	//Alarm Priority setpoint
	{attribute 'OPC.UA.DA' :='1'}
	popa_0082_pt_3119_b_low_priority : INT;
	//Alarm delay setpoint(seconds)
	{attribute 'OPC.UA.DA' :='1'}
	popa_0082_pt_3119_b_low_delay_setpoint : INT;
	//Alarm active for HMI
	{attribute 'OPC.UA.DA' :='1'}
	popa_0082_pt_3119_b_low_active : BOOL;
	//Analog Alarm Setpoint
	{attribute 'OPC.UA.DA' :='1'}
	popa_0082_pt_3119_b_low_setpoint : REAL;
	//Alarm enable
	{attribute 'OPC.UA.DA' :='1'}
	popa_0082_pt_3119_b_low_enable: BOOL;
	
	//Alarm Priority setpoint
	{attribute 'OPC.UA.DA' :='1'}
	popa_0082_pt_3119_b_high_priority : INT;
	//Alarm delay setpoint(seconds)
	{attribute 'OPC.UA.DA' :='1'}
	popa_0082_pt_3119_b_high_delay_setpoint : INT;
	//Alarm active for HMI
	{attribute 'OPC.UA.DA' :='1'}
	popa_0082_pt_3119_b_high_active : BOOL;
	//Analog Alarm Setpoint
	{attribute 'OPC.UA.DA' :='1'}
	popa_0082_pt_3119_b_high_setpoint : REAL;
	//Alarm enable
	{attribute 'OPC.UA.DA' :='1'}
	popa_0082_pt_3119_b_high_enable: BOOL;
	
	//Alarm Priority setpoint
	{attribute 'OPC.UA.DA' :='1'}
	popa_0082_pt_3119_b_high_high_priority : INT;
	//Alarm delay setpoint(seconds)
	{attribute 'OPC.UA.DA' :='1'}
	popa_0082_pt_3119_b_high_high_delay_setpoint : INT;
	//Alarm active for HMI
	{attribute 'OPC.UA.DA' :='1'}
	popa_0082_pt_3119_b_high_high_active : BOOL;
	//Analog Alarm Setpoint
	{attribute 'OPC.UA.DA' :='1'}
	popa_0082_pt_3119_b_high_high_setpoint : REAL;
	//Alarm enable
	{attribute 'OPC.UA.DA' :='1'}
	popa_0082_pt_3119_b_high_high_enable: BOOL;
	
	
	//Raw Min value for analog input
	{attribute 'OPC.UA.DA' :='1'}
	popa_0082_pt_3119_b_raw_min : REAL :=0;
	//Raw max value for analog input
	{attribute 'OPC.UA.DA' :='1'}
	popa_0082_pt_3119_b_raw_max : REAL :=32767;
	//EU Min value for analog input
	{attribute 'OPC.UA.DA' :='1'}
	popa_0082_pt_3119_b_eu_min : REAL;
	//EU Max value for analog input
	{attribute 'OPC.UA.DA' :='1'}
	popa_0082_pt_3119_b_eu_max : REAL;
	//Filter factor value for analog input
	{attribute 'OPC.UA.DA' :='1'}
	popa_0082_pt_3119_b_filter_factor : REAL;
	//Scaled value for analog input
	{attribute 'OPC.UA.DA' :='1'}
	popa_0082_pt_3119_b_scaled_value : REAL;
	
	//---pt_3219-----------------------------------------------------------------------------------------------------------------------
	//Alarm Priority setpoint
	{attribute 'OPC.UA.DA' :='1'}
	popa_0082_pt_3219_b_low_low_priority : INT;
	//Alarm delay setpoint(seconds)
	{attribute 'OPC.UA.DA' :='1'}
	popa_0082_pt_3219_b_low_low_delay_setpoint : INT;
	//Alarm active for HMI
	{attribute 'OPC.UA.DA' :='1'}
	popa_0082_pt_3219_b_low_low_active : BOOL;
	//Analog Alarm Setpoint
	{attribute 'OPC.UA.DA' :='1'}
	popa_0082_pt_3219_b_low_low_setpoint : REAL;
	//Alarm enable
	{attribute 'OPC.UA.DA' :='1'}
	popa_0082_pt_3219_b_low_low_enable: BOOL;
	
	//Alarm Priority setpoint
	{attribute 'OPC.UA.DA' :='1'}
	popa_0082_pt_3219_b_low_priority : INT;
	//Alarm delay setpoint(seconds)
	{attribute 'OPC.UA.DA' :='1'}
	popa_0082_pt_3219_b_low_delay_setpoint : INT;
	//Alarm active for HMI
	{attribute 'OPC.UA.DA' :='1'}
	popa_0082_pt_3219_b_low_active : BOOL;
	//Analog Alarm Setpoint
	{attribute 'OPC.UA.DA' :='1'}
	popa_0082_pt_3219_b_low_setpoint : REAL;
	//Alarm enable
	{attribute 'OPC.UA.DA' :='1'}
	popa_0082_pt_3219_b_low_enable: BOOL;
	
	//Alarm Priority setpoint
	{attribute 'OPC.UA.DA' :='1'}
	popa_0082_pt_3219_b_high_priority : INT;
	//Alarm delay setpoint(seconds)
	{attribute 'OPC.UA.DA' :='1'}
	popa_0082_pt_3219_b_high_delay_setpoint : INT;
	//Alarm active for HMI
	{attribute 'OPC.UA.DA' :='1'}
	popa_0082_pt_3219_b_high_active : BOOL;
	//Analog Alarm Setpoint
	{attribute 'OPC.UA.DA' :='1'}
	popa_0082_pt_3219_b_high_setpoint : REAL;
	//Alarm enable
	{attribute 'OPC.UA.DA' :='1'}
	popa_0082_pt_3219_b_high_enable: BOOL;
	
	//Alarm Priority setpoint
	{attribute 'OPC.UA.DA' :='1'}
	popa_0082_pt_3219_b_high_high_priority : INT;
	//Alarm delay setpoint(seconds)
	{attribute 'OPC.UA.DA' :='1'}
	popa_0082_pt_3219_b_high_high_delay_setpoint : INT;
	//Alarm active for HMI
	{attribute 'OPC.UA.DA' :='1'}
	popa_0082_pt_3219_b_high_high_active : BOOL;
	//Analog Alarm Setpoint
	{attribute 'OPC.UA.DA' :='1'}
	popa_0082_pt_3219_b_high_high_setpoint : REAL;
	//Alarm enable
	{attribute 'OPC.UA.DA' :='1'}
	popa_0082_pt_3219_b_high_high_enable: BOOL;
	
	
	//Raw Min value for analog input
	{attribute 'OPC.UA.DA' :='1'}
	popa_0082_pt_3219_b_raw_min : REAL :=0;
	//Raw max value for analog input
	{attribute 'OPC.UA.DA' :='1'}
	popa_0082_pt_3219_b_raw_max : REAL :=32767;
	//EU Min value for analog input
	{attribute 'OPC.UA.DA' :='1'}
	popa_0082_pt_3219_b_eu_min : REAL;
	//EU Max value for analog input
	{attribute 'OPC.UA.DA' :='1'}
	popa_0082_pt_3219_b_eu_max : REAL;
	//Filter factor value for analog input
	{attribute 'OPC.UA.DA' :='1'}
	popa_0082_pt_3219_b_filter_factor : REAL;
	//Scaled value for analog input
	{attribute 'OPC.UA.DA' :='1'}
	popa_0082_pt_3219_b_scaled_value : REAL;
	
	//---pt_3319-----------------------------------------------------------------------------------------------------------------------
	//Alarm Priority setpoint
	{attribute 'OPC.UA.DA' :='1'}
	popa_0082_pt_3319_b_low_low_priority : INT;
	//Alarm delay setpoint(seconds)
	{attribute 'OPC.UA.DA' :='1'}
	popa_0082_pt_3319_b_low_low_delay_setpoint : INT;
	//Alarm active for HMI
	{attribute 'OPC.UA.DA' :='1'}
	popa_0082_pt_3319_b_low_low_active : BOOL;
	//Analog Alarm Setpoint
	{attribute 'OPC.UA.DA' :='1'}
	popa_0082_pt_3319_b_low_low_setpoint : REAL;
	//Alarm enable
	{attribute 'OPC.UA.DA' :='1'}
	popa_0082_pt_3319_b_low_low_enable: BOOL;
	
	//Alarm Priority setpoint
	{attribute 'OPC.UA.DA' :='1'}
	popa_0082_pt_3319_b_low_priority : INT;
	//Alarm delay setpoint(seconds)
	{attribute 'OPC.UA.DA' :='1'}
	popa_0082_pt_3319_b_low_delay_setpoint : INT;
	//Alarm active for HMI
	{attribute 'OPC.UA.DA' :='1'}
	popa_0082_pt_3319_b_low_active : BOOL;
	//Analog Alarm Setpoint
	{attribute 'OPC.UA.DA' :='1'}
	popa_0082_pt_3319_b_low_setpoint : REAL;
	//Alarm enable
	{attribute 'OPC.UA.DA' :='1'}
	popa_0082_pt_3319_b_low_enable: BOOL;
	
	//Alarm Priority setpoint
	{attribute 'OPC.UA.DA' :='1'}
	popa_0082_pt_3319_b_high_priority : INT;
	//Alarm delay setpoint(seconds)
	{attribute 'OPC.UA.DA' :='1'}
	popa_0082_pt_3319_b_high_delay_setpoint : INT;
	//Alarm active for HMI
	{attribute 'OPC.UA.DA' :='1'}
	popa_0082_pt_3319_b_high_active : BOOL;
	//Analog Alarm Setpoint
	{attribute 'OPC.UA.DA' :='1'}
	popa_0082_pt_3319_b_high_setpoint : REAL;
	//Alarm enable
	{attribute 'OPC.UA.DA' :='1'}
	popa_0082_pt_3319_b_high_enable: BOOL;
	
	//Alarm Priority setpoint
	{attribute 'OPC.UA.DA' :='1'}
	popa_0082_pt_3319_b_high_high_priority : INT;
	//Alarm delay setpoint(seconds)
	{attribute 'OPC.UA.DA' :='1'}
	popa_0082_pt_3319_b_high_high_delay_setpoint : INT;
	//Alarm active for HMI
	{attribute 'OPC.UA.DA' :='1'}
	popa_0082_pt_3319_b_high_high_active : BOOL;
	//Analog Alarm Setpoint
	{attribute 'OPC.UA.DA' :='1'}
	popa_0082_pt_3319_b_high_high_setpoint : REAL;
	//Alarm enable
	{attribute 'OPC.UA.DA' :='1'}
	popa_0082_pt_3319_b_high_high_enable: BOOL;
	
	
	//Raw Min value for analog input
	{attribute 'OPC.UA.DA' :='1'}
	popa_0082_pt_3319_b_raw_min : REAL :=0;
	//Raw max value for analog input
	{attribute 'OPC.UA.DA' :='1'}
	popa_0082_pt_3319_b_raw_max : REAL :=32767;
	//EU Min value for analog input
	{attribute 'OPC.UA.DA' :='1'}
	popa_0082_pt_3319_b_eu_min : REAL;
	//EU Max value for analog input
	{attribute 'OPC.UA.DA' :='1'}
	popa_0082_pt_3319_b_eu_max : REAL;
	//Filter factor value for analog input
	{attribute 'OPC.UA.DA' :='1'}
	popa_0082_pt_3319_b_filter_factor : REAL;
	//Scaled value for analog input
	{attribute 'OPC.UA.DA' :='1'}
	popa_0082_pt_3319_b_scaled_value : REAL;
	
	//---pt_3141-----------------------------------------------------------------------------------------------------------------------
	//Alarm Priority setpoint
	{attribute 'OPC.UA.DA' :='1'}
	popa_0082_pt_3141_b_low_low_priority : INT;
	//Alarm delay setpoint(seconds)
	{attribute 'OPC.UA.DA' :='1'}
	popa_0082_pt_3141_b_low_low_delay_setpoint : INT;
	//Alarm active for HMI
	{attribute 'OPC.UA.DA' :='1'}
	popa_0082_pt_3141_b_low_low_active : BOOL;
	//Analog Alarm Setpoint
	{attribute 'OPC.UA.DA' :='1'}
	popa_0082_pt_3141_b_low_low_setpoint : REAL;
	//Alarm enable
	{attribute 'OPC.UA.DA' :='1'}
	popa_0082_pt_3141_b_low_low_enable: BOOL;
	
	//Alarm Priority setpoint
	{attribute 'OPC.UA.DA' :='1'}
	popa_0082_pt_3141_b_low_priority : INT;
	//Alarm delay setpoint(seconds)
	{attribute 'OPC.UA.DA' :='1'}
	popa_0082_pt_3141_b_low_delay_setpoint : INT;
	//Alarm active for HMI
	{attribute 'OPC.UA.DA' :='1'}
	popa_0082_pt_3141_b_low_active : BOOL;
	//Analog Alarm Setpoint
	{attribute 'OPC.UA.DA' :='1'}
	popa_0082_pt_3141_b_low_setpoint : REAL;
	//Alarm enable
	{attribute 'OPC.UA.DA' :='1'}
	popa_0082_pt_3141_b_low_enable: BOOL;
	
	//Alarm Priority setpoint
	{attribute 'OPC.UA.DA' :='1'}
	popa_0082_pt_3141_b_high_priority : INT;
	//Alarm delay setpoint(seconds)
	{attribute 'OPC.UA.DA' :='1'}
	popa_0082_pt_3141_b_high_delay_setpoint : INT;
	//Alarm active for HMI
	{attribute 'OPC.UA.DA' :='1'}
	popa_0082_pt_3141_b_high_active : BOOL;
	//Analog Alarm Setpoint
	{attribute 'OPC.UA.DA' :='1'}
	popa_0082_pt_3141_b_high_setpoint : REAL;
	//Alarm enable
	{attribute 'OPC.UA.DA' :='1'}
	popa_0082_pt_3141_b_high_enable: BOOL;
	
	//Alarm Priority setpoint
	{attribute 'OPC.UA.DA' :='1'}
	popa_0082_pt_3141_b_high_high_priority : INT;
	//Alarm delay setpoint(seconds)
	{attribute 'OPC.UA.DA' :='1'}
	popa_0082_pt_3141_b_high_high_delay_setpoint : INT;
	//Alarm active for HMI
	{attribute 'OPC.UA.DA' :='1'}
	popa_0082_pt_3141_b_high_high_active : BOOL;
	//Analog Alarm Setpoint
	{attribute 'OPC.UA.DA' :='1'}
	popa_0082_pt_3141_b_high_high_setpoint : REAL;
	//Alarm enable
	{attribute 'OPC.UA.DA' :='1'}
	popa_0082_pt_3141_b_high_high_enable: BOOL;
	
	
	//Raw Min value for analog input
	{attribute 'OPC.UA.DA' :='1'}
	popa_0082_pt_3141_b_raw_min : REAL :=0;
	//Raw max value for analog input
	{attribute 'OPC.UA.DA' :='1'}
	popa_0082_pt_3141_b_raw_max : REAL :=32767;
	//EU Min value for analog input
	{attribute 'OPC.UA.DA' :='1'}
	popa_0082_pt_3141_b_eu_min : REAL;
	//EU Max value for analog input
	{attribute 'OPC.UA.DA' :='1'}
	popa_0082_pt_3141_b_eu_max : REAL;
	//Filter factor value for analog input
	{attribute 'OPC.UA.DA' :='1'}
	popa_0082_pt_3141_b_filter_factor : REAL;
	//Scaled value for analog input
	{attribute 'OPC.UA.DA' :='1'}
	popa_0082_pt_3141_b_scaled_value : REAL;
	
	//---pt_3241-----------------------------------------------------------------------------------------------------------------------
	//Alarm Priority setpoint
	{attribute 'OPC.UA.DA' :='1'}
	popa_0082_pt_3241_b_low_low_priority : INT;
	//Alarm delay setpoint(seconds)
	{attribute 'OPC.UA.DA' :='1'}
	popa_0082_pt_3241_b_low_low_delay_setpoint : INT;
	//Alarm active for HMI
	{attribute 'OPC.UA.DA' :='1'}
	popa_0082_pt_3241_b_low_low_active : BOOL;
	//Analog Alarm Setpoint
	{attribute 'OPC.UA.DA' :='1'}
	popa_0082_pt_3241_b_low_low_setpoint : REAL;
	//Alarm enable
	{attribute 'OPC.UA.DA' :='1'}
	popa_0082_pt_3241_b_low_low_enable: BOOL;
	
	//Alarm Priority setpoint
	{attribute 'OPC.UA.DA' :='1'}
	popa_0082_pt_3241_b_low_priority : INT;
	//Alarm delay setpoint(seconds)
	{attribute 'OPC.UA.DA' :='1'}
	popa_0082_pt_3241_b_low_delay_setpoint : INT;
	//Alarm active for HMI
	{attribute 'OPC.UA.DA' :='1'}
	popa_0082_pt_3241_b_low_active : BOOL;
	//Analog Alarm Setpoint
	{attribute 'OPC.UA.DA' :='1'}
	popa_0082_pt_3241_b_low_setpoint : REAL;
	//Alarm enable
	{attribute 'OPC.UA.DA' :='1'}
	popa_0082_pt_3241_b_low_enable: BOOL;
	
	//Alarm Priority setpoint
	{attribute 'OPC.UA.DA' :='1'}
	popa_0082_pt_3241_b_high_priority : INT;
	//Alarm delay setpoint(seconds)
	{attribute 'OPC.UA.DA' :='1'}
	popa_0082_pt_3241_b_high_delay_setpoint : INT;
	//Alarm active for HMI
	{attribute 'OPC.UA.DA' :='1'}
	popa_0082_pt_3241_b_high_active : BOOL;
	//Analog Alarm Setpoint
	{attribute 'OPC.UA.DA' :='1'}
	popa_0082_pt_3241_b_high_setpoint : REAL;
	//Alarm enable
	{attribute 'OPC.UA.DA' :='1'}
	popa_0082_pt_3241_b_high_enable: BOOL;
	
	//Alarm Priority setpoint
	{attribute 'OPC.UA.DA' :='1'}
	popa_0082_pt_3241_b_high_high_priority : INT;
	//Alarm delay setpoint(seconds)
	{attribute 'OPC.UA.DA' :='1'}
	popa_0082_pt_3241_b_high_high_delay_setpoint : INT;
	//Alarm active for HMI
	{attribute 'OPC.UA.DA' :='1'}
	popa_0082_pt_3241_b_high_high_active : BOOL;
	//Analog Alarm Setpoint
	{attribute 'OPC.UA.DA' :='1'}
	popa_0082_pt_3241_b_high_high_setpoint : REAL;
	//Alarm enable
	{attribute 'OPC.UA.DA' :='1'}
	popa_0082_pt_3241_b_high_high_enable: BOOL;
	
	
	//Raw Min value for analog input
	{attribute 'OPC.UA.DA' :='1'}
	popa_0082_pt_3241_b_raw_min : REAL :=0;
	//Raw max value for analog input
	{attribute 'OPC.UA.DA' :='1'}
	popa_0082_pt_3241_b_raw_max : REAL :=32767;
	//EU Min value for analog input
	{attribute 'OPC.UA.DA' :='1'}
	popa_0082_pt_3241_b_eu_min : REAL;
	//EU Max value for analog input
	{attribute 'OPC.UA.DA' :='1'}
	popa_0082_pt_3241_b_eu_max : REAL;
	//Filter factor value for analog input
	{attribute 'OPC.UA.DA' :='1'}
	popa_0082_pt_3241_b_filter_factor : REAL;
	//Scaled value for analog input
	{attribute 'OPC.UA.DA' :='1'}
	popa_0082_pt_3241_b_scaled_value : REAL;
	
	//---pt_3341-----------------------------------------------------------------------------------------------------------------------
	//Alarm Priority setpoint
	{attribute 'OPC.UA.DA' :='1'}
	popa_0082_pt_3341_b_low_low_priority : INT;
	//Alarm delay setpoint(seconds)
	{attribute 'OPC.UA.DA' :='1'}
	popa_0082_pt_3341_b_low_low_delay_setpoint : INT;
	//Alarm active for HMI
	{attribute 'OPC.UA.DA' :='1'}
	popa_0082_pt_3341_b_low_low_active : BOOL;
	//Analog Alarm Setpoint
	{attribute 'OPC.UA.DA' :='1'}
	popa_0082_pt_3341_b_low_low_setpoint : REAL;
	//Alarm enable
	{attribute 'OPC.UA.DA' :='1'}
	popa_0082_pt_3341_b_low_low_enable: BOOL;
	
	//Alarm Priority setpoint
	{attribute 'OPC.UA.DA' :='1'}
	popa_0082_pt_3341_b_low_priority : INT;
	//Alarm delay setpoint(seconds)
	{attribute 'OPC.UA.DA' :='1'}
	popa_0082_pt_3341_b_low_delay_setpoint : INT;
	//Alarm active for HMI
	{attribute 'OPC.UA.DA' :='1'}
	popa_0082_pt_3341_b_low_active : BOOL;
	//Analog Alarm Setpoint
	{attribute 'OPC.UA.DA' :='1'}
	popa_0082_pt_3341_b_low_setpoint : REAL;
	//Alarm enable
	{attribute 'OPC.UA.DA' :='1'}
	popa_0082_pt_3341_b_low_enable: BOOL;
	
	//Alarm Priority setpoint
	{attribute 'OPC.UA.DA' :='1'}
	popa_0082_pt_3341_b_high_priority : INT;
	//Alarm delay setpoint(seconds)
	{attribute 'OPC.UA.DA' :='1'}
	popa_0082_pt_3341_b_high_delay_setpoint : INT;
	//Alarm active for HMI
	{attribute 'OPC.UA.DA' :='1'}
	popa_0082_pt_3341_b_high_active : BOOL;
	//Analog Alarm Setpoint
	{attribute 'OPC.UA.DA' :='1'}
	popa_0082_pt_3341_b_high_setpoint : REAL;
	//Alarm enable
	{attribute 'OPC.UA.DA' :='1'}
	popa_0082_pt_3341_b_high_enable: BOOL;
	
	//Alarm Priority setpoint
	{attribute 'OPC.UA.DA' :='1'}
	popa_0082_pt_3341_b_high_high_priority : INT;
	//Alarm delay setpoint(seconds)
	{attribute 'OPC.UA.DA' :='1'}
	popa_0082_pt_3341_b_high_high_delay_setpoint : INT;
	//Alarm active for HMI
	{attribute 'OPC.UA.DA' :='1'}
	popa_0082_pt_3341_b_high_high_active : BOOL;
	//Analog Alarm Setpoint
	{attribute 'OPC.UA.DA' :='1'}
	popa_0082_pt_3341_b_high_high_setpoint : REAL;
	//Alarm enable
	{attribute 'OPC.UA.DA' :='1'}
	popa_0082_pt_3341_b_high_high_enable: BOOL;
	
	
	//Raw Min value for analog input
	{attribute 'OPC.UA.DA' :='1'}
	popa_0082_pt_3341_b_raw_min : REAL :=0;
	//Raw max value for analog input
	{attribute 'OPC.UA.DA' :='1'}
	popa_0082_pt_3341_b_raw_max : REAL :=32767;
	//EU Min value for analog input
	{attribute 'OPC.UA.DA' :='1'}
	popa_0082_pt_3341_b_eu_min : REAL;
	//EU Max value for analog input
	{attribute 'OPC.UA.DA' :='1'}
	popa_0082_pt_3341_b_eu_max : REAL;
	//Filter factor value for analog input
	{attribute 'OPC.UA.DA' :='1'}
	popa_0082_pt_3341_b_filter_factor : REAL;
	//Scaled value for analog input
	{attribute 'OPC.UA.DA' :='1'}
	popa_0082_pt_3341_b_scaled_value : REAL;
	
//---pt_3428-----------------------------------------------------------------------------------------------------------------------
	//Alarm Priority setpoint
	{attribute 'OPC.UA.DA' :='1'}
	popa_0092_pt_3428_b_low_low_priority : INT;
	//Alarm delay setpoint(seconds)
	{attribute 'OPC.UA.DA' :='1'}
	popa_0092_pt_3428_b_low_low_delay_setpoint : INT;
	//Alarm active for HMI
	{attribute 'OPC.UA.DA' :='1'}
	popa_0092_pt_3428_b_low_low_active : BOOL;
	//Analog Alarm Setpoint
	{attribute 'OPC.UA.DA' :='1'}
	popa_0092_pt_3428_b_low_low_setpoint : REAL;
	//Alarm enable
	{attribute 'OPC.UA.DA' :='1'}
	popa_0092_pt_3428_b_low_low_enable: BOOL;
	
	//Alarm Priority setpoint
	{attribute 'OPC.UA.DA' :='1'}
	popa_0092_pt_3428_b_low_priority : INT;
	//Alarm delay setpoint(seconds)
	{attribute 'OPC.UA.DA' :='1'}
	popa_0092_pt_3428_b_low_delay_setpoint : INT;
	//Alarm active for HMI
	{attribute 'OPC.UA.DA' :='1'}
	popa_0092_pt_3428_b_low_active : BOOL;
	//Analog Alarm Setpoint
	{attribute 'OPC.UA.DA' :='1'}
	popa_0092_pt_3428_b_low_setpoint : REAL;
	//Alarm enable
	{attribute 'OPC.UA.DA' :='1'}
	popa_0092_pt_3428_b_low_enable: BOOL;
	
	//Alarm Priority setpoint
	{attribute 'OPC.UA.DA' :='1'}
	popa_0092_pt_3428_b_high_priority : INT;
	//Alarm delay setpoint(seconds)
	{attribute 'OPC.UA.DA' :='1'}
	popa_0092_pt_3428_b_high_delay_setpoint : INT;
	//Alarm active for HMI
	{attribute 'OPC.UA.DA' :='1'}
	popa_0092_pt_3428_b_high_active : BOOL;
	//Analog Alarm Setpoint
	{attribute 'OPC.UA.DA' :='1'}
	popa_0092_pt_3428_b_high_setpoint : REAL;
	//Alarm enable
	{attribute 'OPC.UA.DA' :='1'}
	popa_0092_pt_3428_b_high_enable: BOOL;
	
	//Alarm Priority setpoint
	{attribute 'OPC.UA.DA' :='1'}
	popa_0092_pt_3428_b_high_high_priority : INT;
	//Alarm delay setpoint(seconds)
	{attribute 'OPC.UA.DA' :='1'}
	popa_0092_pt_3428_b_high_high_delay_setpoint : INT;
	//Alarm active for HMI
	{attribute 'OPC.UA.DA' :='1'}
	popa_0092_pt_3428_b_high_high_active : BOOL;
	//Analog Alarm Setpoint
	{attribute 'OPC.UA.DA' :='1'}
	popa_0092_pt_3428_b_high_high_setpoint : REAL;
	//Alarm enable
	{attribute 'OPC.UA.DA' :='1'}
	popa_0092_pt_3428_b_high_high_enable: BOOL;
	
	
	//Raw Min value for analog input
	{attribute 'OPC.UA.DA' :='1'}
	popa_0092_pt_3428_b_raw_min : REAL :=0;
	//Raw max value for analog input
	{attribute 'OPC.UA.DA' :='1'}
	popa_0092_pt_3428_b_raw_max : REAL :=32767;
	//EU Min value for analog input
	{attribute 'OPC.UA.DA' :='1'}
	popa_0092_pt_3428_b_eu_min : REAL;
	//EU Max value for analog input
	{attribute 'OPC.UA.DA' :='1'}
	popa_0092_pt_3428_b_eu_max : REAL;
	//Filter factor value for analog input
	{attribute 'OPC.UA.DA' :='1'}
	popa_0092_pt_3428_b_filter_factor : REAL;
	//Scaled value for analog input
	{attribute 'OPC.UA.DA' :='1'}
	popa_0092_pt_3428_b_scaled_value : REAL;
	
	//---pt_3414-----------------------------------------------------------------------------------------------------------------------
	//Alarm Priority setpoint
	{attribute 'OPC.UA.DA' :='1'}
	popa_0092_pt_3414_b_low_low_priority : INT;
	//Alarm delay setpoint(seconds)
	{attribute 'OPC.UA.DA' :='1'}
	popa_0092_pt_3414_b_low_low_delay_setpoint : INT;
	//Alarm active for HMI
	{attribute 'OPC.UA.DA' :='1'}
	popa_0092_pt_3414_b_low_low_active : BOOL;
	//Analog Alarm Setpoint
	{attribute 'OPC.UA.DA' :='1'}
	popa_0092_pt_3414_b_low_low_setpoint : REAL;
	//Alarm enable
	{attribute 'OPC.UA.DA' :='1'}
	popa_0092_pt_3414_b_low_low_enable: BOOL;
	
	//Alarm Priority setpoint
	{attribute 'OPC.UA.DA' :='1'}
	popa_0092_pt_3414_b_low_priority : INT;
	//Alarm delay setpoint(seconds)
	{attribute 'OPC.UA.DA' :='1'}
	popa_0092_pt_3414_b_low_delay_setpoint : INT;
	//Alarm active for HMI
	{attribute 'OPC.UA.DA' :='1'}
	popa_0092_pt_3414_b_low_active : BOOL;
	//Analog Alarm Setpoint
	{attribute 'OPC.UA.DA' :='1'}
	popa_0092_pt_3414_b_low_setpoint : REAL;
	//Alarm enable
	{attribute 'OPC.UA.DA' :='1'}
	popa_0092_pt_3414_b_low_enable: BOOL;
	
	//Alarm Priority setpoint
	{attribute 'OPC.UA.DA' :='1'}
	popa_0092_pt_3414_b_high_priority : INT;
	//Alarm delay setpoint(seconds)
	{attribute 'OPC.UA.DA' :='1'}
	popa_0092_pt_3414_b_high_delay_setpoint : INT;
	//Alarm active for HMI
	{attribute 'OPC.UA.DA' :='1'}
	popa_0092_pt_3414_b_high_active : BOOL;
	//Analog Alarm Setpoint
	{attribute 'OPC.UA.DA' :='1'}
	popa_0092_pt_3414_b_high_setpoint : REAL;
	//Alarm enable
	{attribute 'OPC.UA.DA' :='1'}
	popa_0092_pt_3414_b_high_enable: BOOL;
	
	//Alarm Priority setpoint
	{attribute 'OPC.UA.DA' :='1'}
	popa_0092_pt_3414_b_high_high_priority : INT;
	//Alarm delay setpoint(seconds)
	{attribute 'OPC.UA.DA' :='1'}
	popa_0092_pt_3414_b_high_high_delay_setpoint : INT;
	//Alarm active for HMI
	{attribute 'OPC.UA.DA' :='1'}
	popa_0092_pt_3414_b_high_high_active : BOOL;
	//Analog Alarm Setpoint
	{attribute 'OPC.UA.DA' :='1'}
	popa_0092_pt_3414_b_high_high_setpoint : REAL;
	//Alarm enable
	{attribute 'OPC.UA.DA' :='1'}
	popa_0092_pt_3414_b_high_high_enable: BOOL;
	
	
	//Raw Min value for analog input
	{attribute 'OPC.UA.DA' :='1'}
	popa_0092_pt_3414_b_raw_min : REAL :=0;
	//Raw max value for analog input
	{attribute 'OPC.UA.DA' :='1'}
	popa_0092_pt_3414_b_raw_max : REAL :=32767;
	//EU Min value for analog input
	{attribute 'OPC.UA.DA' :='1'}
	popa_0092_pt_3414_b_eu_min : REAL;
	//EU Max value for analog input
	{attribute 'OPC.UA.DA' :='1'}
	popa_0092_pt_3414_b_eu_max : REAL;
	//Filter factor value for analog input
	{attribute 'OPC.UA.DA' :='1'}
	popa_0092_pt_3414_b_filter_factor : REAL;
	//Scaled value for analog input
	{attribute 'OPC.UA.DA' :='1'}
	popa_0092_pt_3414_b_scaled_value : REAL;
	
	//---tt_3118-----------------------------------------------------------------------------------------------------------------------
	//Alarm Priority setpoint
	{attribute 'OPC.UA.DA' :='1'}
	popa_0082_tt_3118_b_low_low_priority : INT;
	//Alarm delay setpoint(seconds)
	{attribute 'OPC.UA.DA' :='1'}
	popa_0082_tt_3118_b_low_low_delay_setpoint : INT;
	//Alarm active for HMI
	{attribute 'OPC.UA.DA' :='1'}
	popa_0082_tt_3118_b_low_low_active : BOOL;
	//Analog Alarm Setpoint
	{attribute 'OPC.UA.DA' :='1'}
	popa_0082_tt_3118_b_low_low_setpoint : REAL;
	//Alarm enable
	{attribute 'OPC.UA.DA' :='1'}
	popa_0082_tt_3118_b_low_low_enable: BOOL;
	
	//Alarm Priority setpoint
	{attribute 'OPC.UA.DA' :='1'}
	popa_0082_tt_3118_b_low_priority : INT;
	//Alarm delay setpoint(seconds)
	{attribute 'OPC.UA.DA' :='1'}
	popa_0082_tt_3118_b_low_delay_setpoint : INT;
	//Alarm active for HMI
	{attribute 'OPC.UA.DA' :='1'}
	popa_0082_tt_3118_b_low_active : BOOL;
	//Analog Alarm Setpoint
	{attribute 'OPC.UA.DA' :='1'}
	popa_0082_tt_3118_b_low_setpoint : REAL;
	//Alarm enable
	{attribute 'OPC.UA.DA' :='1'}
	popa_0082_tt_3118_b_low_enable: BOOL;
	
	//Alarm Priority setpoint
	{attribute 'OPC.UA.DA' :='1'}
	popa_0082_tt_3118_b_high_priority : INT;
	//Alarm delay setpoint(seconds)
	{attribute 'OPC.UA.DA' :='1'}
	popa_0082_tt_3118_b_high_delay_setpoint : INT;
	//Alarm active for HMI
	{attribute 'OPC.UA.DA' :='1'}
	popa_0082_tt_3118_b_high_active : BOOL;
	//Analog Alarm Setpoint
	{attribute 'OPC.UA.DA' :='1'}
	popa_0082_tt_3118_b_high_setpoint : REAL;
	//Alarm enable
	{attribute 'OPC.UA.DA' :='1'}
	popa_0082_tt_3118_b_high_enable: BOOL;
	
	//Alarm Priority setpoint
	{attribute 'OPC.UA.DA' :='1'}
	popa_0082_tt_3118_b_high_high_priority : INT;
	//Alarm delay setpoint(seconds)
	{attribute 'OPC.UA.DA' :='1'}
	popa_0082_tt_3118_b_high_high_delay_setpoint : INT;
	//Alarm active for HMI
	{attribute 'OPC.UA.DA' :='1'}
	popa_0082_tt_3118_b_high_high_active : BOOL;
	//Analog Alarm Setpoint
	{attribute 'OPC.UA.DA' :='1'}
	popa_0082_tt_3118_b_high_high_setpoint : REAL;
	//Alarm enable
	{attribute 'OPC.UA.DA' :='1'}
	popa_0082_tt_3118_b_high_high_enable: BOOL;
	
	
	//Raw Min value for analog input
	{attribute 'OPC.UA.DA' :='1'}
	popa_0082_tt_3118_b_raw_min : REAL :=0;
	//Raw max value for analog input
	{attribute 'OPC.UA.DA' :='1'}
	popa_0082_tt_3118_b_raw_max : REAL :=32767;
	//EU Min value for analog input
	{attribute 'OPC.UA.DA' :='1'}
	popa_0082_tt_3118_b_eu_min : REAL;
	//EU Max value for analog input
	{attribute 'OPC.UA.DA' :='1'}
	popa_0082_tt_3118_b_eu_max : REAL;
	//Filter factor value for analog input
	{attribute 'OPC.UA.DA' :='1'}
	popa_0082_tt_3118_b_filter_factor : REAL;
	//Scaled value for analog input
	{attribute 'OPC.UA.DA' :='1'}
	popa_0082_tt_3118_b_scaled_value : REAL;
	
	//---tt_3218-----------------------------------------------------------------------------------------------------------------------
	//Alarm Priority setpoint
	{attribute 'OPC.UA.DA' :='1'}
	popa_0082_tt_3218_b_low_low_priority : INT;
	//Alarm delay setpoint(seconds)
	{attribute 'OPC.UA.DA' :='1'}
	popa_0082_tt_3218_b_low_low_delay_setpoint : INT;
	//Alarm active for HMI
	{attribute 'OPC.UA.DA' :='1'}
	popa_0082_tt_3218_b_low_low_active : BOOL;
	//Analog Alarm Setpoint
	{attribute 'OPC.UA.DA' :='1'}
	popa_0082_tt_3218_b_low_low_setpoint : REAL;
	//Alarm enable
	{attribute 'OPC.UA.DA' :='1'}
	popa_0082_tt_3218_b_low_low_enable: BOOL;
	
	//Alarm Priority setpoint
	{attribute 'OPC.UA.DA' :='1'}
	popa_0082_tt_3218_b_low_priority : INT;
	//Alarm delay setpoint(seconds)
	{attribute 'OPC.UA.DA' :='1'}
	popa_0082_tt_3218_b_low_delay_setpoint : INT;
	//Alarm active for HMI
	{attribute 'OPC.UA.DA' :='1'}
	popa_0082_tt_3218_b_low_active : BOOL;
	//Analog Alarm Setpoint
	{attribute 'OPC.UA.DA' :='1'}
	popa_0082_tt_3218_b_low_setpoint : REAL;
	//Alarm enable
	{attribute 'OPC.UA.DA' :='1'}
	popa_0082_tt_3218_b_low_enable: BOOL;
	
	//Alarm Priority setpoint
	{attribute 'OPC.UA.DA' :='1'}
	popa_0082_tt_3218_b_high_priority : INT;
	//Alarm delay setpoint(seconds)
	{attribute 'OPC.UA.DA' :='1'}
	popa_0082_tt_3218_b_high_delay_setpoint : INT;
	//Alarm active for HMI
	{attribute 'OPC.UA.DA' :='1'}
	popa_0082_tt_3218_b_high_active : BOOL;
	//Analog Alarm Setpoint
	{attribute 'OPC.UA.DA' :='1'}
	popa_0082_tt_3218_b_high_setpoint : REAL;
	//Alarm enable
	{attribute 'OPC.UA.DA' :='1'}
	popa_0082_tt_3218_b_high_enable: BOOL;
	
	//Alarm Priority setpoint
	{attribute 'OPC.UA.DA' :='1'}
	popa_0082_tt_3218_b_high_high_priority : INT;
	//Alarm delay setpoint(seconds)
	{attribute 'OPC.UA.DA' :='1'}
	popa_0082_tt_3218_b_high_high_delay_setpoint : INT;
	//Alarm active for HMI
	{attribute 'OPC.UA.DA' :='1'}
	popa_0082_tt_3218_b_high_high_active : BOOL;
	//Analog Alarm Setpoint
	{attribute 'OPC.UA.DA' :='1'}
	popa_0082_tt_3218_b_high_high_setpoint : REAL;
	//Alarm enable
	{attribute 'OPC.UA.DA' :='1'}
	popa_0082_tt_3218_b_high_high_enable: BOOL;
	
	
	//Raw Min value for analog input
	{attribute 'OPC.UA.DA' :='1'}
	popa_0082_tt_3218_b_raw_min : REAL :=0;
	//Raw max value for analog input
	{attribute 'OPC.UA.DA' :='1'}
	popa_0082_tt_3218_b_raw_max : REAL :=32767;
	//EU Min value for analog input
	{attribute 'OPC.UA.DA' :='1'}
	popa_0082_tt_3218_b_eu_min : REAL;
	//EU Max value for analog input
	{attribute 'OPC.UA.DA' :='1'}
	popa_0082_tt_3218_b_eu_max : REAL;
	//Filter factor value for analog input
	{attribute 'OPC.UA.DA' :='1'}
	popa_0082_tt_3218_b_filter_factor : REAL;
	//Scaled value for analog input
	{attribute 'OPC.UA.DA' :='1'}
	popa_0082_tt_3218_b_scaled_value : REAL;
	
	//---tt_3318-----------------------------------------------------------------------------------------------------------------------
	//Alarm Priority setpoint
	{attribute 'OPC.UA.DA' :='1'}
	popa_0082_tt_3318_b_low_low_priority : INT;
	//Alarm delay setpoint(seconds)
	{attribute 'OPC.UA.DA' :='1'}
	popa_0082_tt_3318_b_low_low_delay_setpoint : INT;
	//Alarm active for HMI
	{attribute 'OPC.UA.DA' :='1'}
	popa_0082_tt_3318_b_low_low_active : BOOL;
	//Analog Alarm Setpoint
	{attribute 'OPC.UA.DA' :='1'}
	popa_0082_tt_3318_b_low_low_setpoint : REAL;
	//Alarm enable
	{attribute 'OPC.UA.DA' :='1'}
	popa_0082_tt_3318_b_low_low_enable: BOOL;
	
	//Alarm Priority setpoint
	{attribute 'OPC.UA.DA' :='1'}
	popa_0082_tt_3318_b_low_priority : INT;
	//Alarm delay setpoint(seconds)
	{attribute 'OPC.UA.DA' :='1'}
	popa_0082_tt_3318_b_low_delay_setpoint : INT;
	//Alarm active for HMI
	{attribute 'OPC.UA.DA' :='1'}
	popa_0082_tt_3318_b_low_active : BOOL;
	//Analog Alarm Setpoint
	{attribute 'OPC.UA.DA' :='1'}
	popa_0082_tt_3318_b_low_setpoint : REAL;
	//Alarm enable
	{attribute 'OPC.UA.DA' :='1'}
	popa_0082_tt_3318_b_low_enable: BOOL;
	
	//Alarm Priority setpoint
	{attribute 'OPC.UA.DA' :='1'}
	popa_0082_tt_3318_b_high_priority : INT;
	//Alarm delay setpoint(seconds)
	{attribute 'OPC.UA.DA' :='1'}
	popa_0082_tt_3318_b_high_delay_setpoint : INT;
	//Alarm active for HMI
	{attribute 'OPC.UA.DA' :='1'}
	popa_0082_tt_3318_b_high_active : BOOL;
	//Analog Alarm Setpoint
	{attribute 'OPC.UA.DA' :='1'}
	popa_0082_tt_3318_b_high_setpoint : REAL;
	//Alarm enable
	{attribute 'OPC.UA.DA' :='1'}
	popa_0082_tt_3318_b_high_enable: BOOL;
	
	//Alarm Priority setpoint
	{attribute 'OPC.UA.DA' :='1'}
	popa_0082_tt_3318_b_high_high_priority : INT;
	//Alarm delay setpoint(seconds)
	{attribute 'OPC.UA.DA' :='1'}
	popa_0082_tt_3318_b_high_high_delay_setpoint : INT;
	//Alarm active for HMI
	{attribute 'OPC.UA.DA' :='1'}
	popa_0082_tt_3318_b_high_high_active : BOOL;
	//Analog Alarm Setpoint
	{attribute 'OPC.UA.DA' :='1'}
	popa_0082_tt_3318_b_high_high_setpoint : REAL;
	//Alarm enable
	{attribute 'OPC.UA.DA' :='1'}
	popa_0082_tt_3318_b_high_high_enable: BOOL;
	
	
	//Raw Min value for analog input
	{attribute 'OPC.UA.DA' :='1'}
	popa_0082_tt_3318_b_raw_min : REAL :=0;
	//Raw max value for analog input
	{attribute 'OPC.UA.DA' :='1'}
	popa_0082_tt_3318_b_raw_max : REAL :=32767;
	//EU Min value for analog input
	{attribute 'OPC.UA.DA' :='1'}
	popa_0082_tt_3318_b_eu_min : REAL;
	//EU Max value for analog input
	{attribute 'OPC.UA.DA' :='1'}
	popa_0082_tt_3318_b_eu_max : REAL;
	//Filter factor value for analog input
	{attribute 'OPC.UA.DA' :='1'}
	popa_0082_tt_3318_b_filter_factor : REAL;
	//Scaled value for analog input
	{attribute 'OPC.UA.DA' :='1'}
	popa_0082_tt_3318_b_scaled_value : REAL;
	
	//---tt_3140-----------------------------------------------------------------------------------------------------------------------
	//Alarm Priority setpoint
	{attribute 'OPC.UA.DA' :='1'}
	popa_0082_tt_3140_b_low_low_priority : INT;
	//Alarm delay setpoint(seconds)
	{attribute 'OPC.UA.DA' :='1'}
	popa_0082_tt_3140_b_low_low_delay_setpoint : INT;
	//Alarm active for HMI
	{attribute 'OPC.UA.DA' :='1'}
	popa_0082_tt_3140_b_low_low_active : BOOL;
	//Analog Alarm Setpoint
	{attribute 'OPC.UA.DA' :='1'}
	popa_0082_tt_3140_b_low_low_setpoint : REAL;
	//Alarm enable
	{attribute 'OPC.UA.DA' :='1'}
	popa_0082_tt_3140_b_low_low_enable: BOOL;
	
	//Alarm Priority setpoint
	{attribute 'OPC.UA.DA' :='1'}
	popa_0082_tt_3140_b_low_priority : INT;
	//Alarm delay setpoint(seconds)
	{attribute 'OPC.UA.DA' :='1'}
	popa_0082_tt_3140_b_low_delay_setpoint : INT;
	//Alarm active for HMI
	{attribute 'OPC.UA.DA' :='1'}
	popa_0082_tt_3140_b_low_active : BOOL;
	//Analog Alarm Setpoint
	{attribute 'OPC.UA.DA' :='1'}
	popa_0082_tt_3140_b_low_setpoint : REAL;
	//Alarm enable
	{attribute 'OPC.UA.DA' :='1'}
	popa_0082_tt_3140_b_low_enable: BOOL;
	
	//Alarm Priority setpoint
	{attribute 'OPC.UA.DA' :='1'}
	popa_0082_tt_3140_b_high_priority : INT;
	//Alarm delay setpoint(seconds)
	{attribute 'OPC.UA.DA' :='1'}
	popa_0082_tt_3140_b_high_delay_setpoint : INT;
	//Alarm active for HMI
	{attribute 'OPC.UA.DA' :='1'}
	popa_0082_tt_3140_b_high_active : BOOL;
	//Analog Alarm Setpoint
	{attribute 'OPC.UA.DA' :='1'}
	popa_0082_tt_3140_b_high_setpoint : REAL;
	//Alarm enable
	{attribute 'OPC.UA.DA' :='1'}
	popa_0082_tt_3140_b_high_enable: BOOL;
	
	//Alarm Priority setpoint
	{attribute 'OPC.UA.DA' :='1'}
	popa_0082_tt_3140_b_high_high_priority : INT;
	//Alarm delay setpoint(seconds)
	{attribute 'OPC.UA.DA' :='1'}
	popa_0082_tt_3140_b_high_high_delay_setpoint : INT;
	//Alarm active for HMI
	{attribute 'OPC.UA.DA' :='1'}
	popa_0082_tt_3140_b_high_high_active : BOOL;
	//Analog Alarm Setpoint
	{attribute 'OPC.UA.DA' :='1'}
	popa_0082_tt_3140_b_high_high_setpoint : REAL;
	//Alarm enable
	{attribute 'OPC.UA.DA' :='1'}
	popa_0082_tt_3140_b_high_high_enable: BOOL;
	
	
	//Raw Min value for analog input
	{attribute 'OPC.UA.DA' :='1'}
	popa_0082_tt_3140_b_raw_min : REAL :=0;
	//Raw max value for analog input
	{attribute 'OPC.UA.DA' :='1'}
	popa_0082_tt_3140_b_raw_max : REAL :=32767;
	//EU Min value for analog input
	{attribute 'OPC.UA.DA' :='1'}
	popa_0082_tt_3140_b_eu_min : REAL;
	//EU Max value for analog input
	{attribute 'OPC.UA.DA' :='1'}
	popa_0082_tt_3140_b_eu_max : REAL;
	//Filter factor value for analog input
	{attribute 'OPC.UA.DA' :='1'}
	popa_0082_tt_3140_b_filter_factor : REAL;
	//Scaled value for analog input
	{attribute 'OPC.UA.DA' :='1'}
	popa_0082_tt_3140_b_scaled_value : REAL;
	
	//---tt_3240-----------------------------------------------------------------------------------------------------------------------
	//Alarm Priority setpoint
	{attribute 'OPC.UA.DA' :='1'}
	popa_0082_tt_3240_b_low_low_priority : INT;
	//Alarm delay setpoint(seconds)
	{attribute 'OPC.UA.DA' :='1'}
	popa_0082_tt_3240_b_low_low_delay_setpoint : INT;
	//Alarm active for HMI
	{attribute 'OPC.UA.DA' :='1'}
	popa_0082_tt_3240_b_low_low_active : BOOL;
	//Analog Alarm Setpoint
	{attribute 'OPC.UA.DA' :='1'}
	popa_0082_tt_3240_b_low_low_setpoint : REAL;
	//Alarm enable
	{attribute 'OPC.UA.DA' :='1'}
	popa_0082_tt_3240_b_low_low_enable: BOOL;
	
	//Alarm Priority setpoint
	{attribute 'OPC.UA.DA' :='1'}
	popa_0082_tt_3240_b_low_priority : INT;
	//Alarm delay setpoint(seconds)
	{attribute 'OPC.UA.DA' :='1'}
	popa_0082_tt_3240_b_low_delay_setpoint : INT;
	//Alarm active for HMI
	{attribute 'OPC.UA.DA' :='1'}
	popa_0082_tt_3240_b_low_active : BOOL;
	//Analog Alarm Setpoint
	{attribute 'OPC.UA.DA' :='1'}
	popa_0082_tt_3240_b_low_setpoint : REAL;
	//Alarm enable
	{attribute 'OPC.UA.DA' :='1'}
	popa_0082_tt_3240_b_low_enable: BOOL;
	
	//Alarm Priority setpoint
	{attribute 'OPC.UA.DA' :='1'}
	popa_0082_tt_3240_b_high_priority : INT;
	//Alarm delay setpoint(seconds)
	{attribute 'OPC.UA.DA' :='1'}
	popa_0082_tt_3240_b_high_delay_setpoint : INT;
	//Alarm active for HMI
	{attribute 'OPC.UA.DA' :='1'}
	popa_0082_tt_3240_b_high_active : BOOL;
	//Analog Alarm Setpoint
	{attribute 'OPC.UA.DA' :='1'}
	popa_0082_tt_3240_b_high_setpoint : REAL;
	//Alarm enable
	{attribute 'OPC.UA.DA' :='1'}
	popa_0082_tt_3240_b_high_enable: BOOL;
	
	//Alarm Priority setpoint
	{attribute 'OPC.UA.DA' :='1'}
	popa_0082_tt_3240_b_high_high_priority : INT;
	//Alarm delay setpoint(seconds)
	{attribute 'OPC.UA.DA' :='1'}
	popa_0082_tt_3240_b_high_high_delay_setpoint : INT;
	//Alarm active for HMI
	{attribute 'OPC.UA.DA' :='1'}
	popa_0082_tt_3240_b_high_high_active : BOOL;
	//Analog Alarm Setpoint
	{attribute 'OPC.UA.DA' :='1'}
	popa_0082_tt_3240_b_high_high_setpoint : REAL;
	//Alarm enable
	{attribute 'OPC.UA.DA' :='1'}
	popa_0082_tt_3240_b_high_high_enable: BOOL;
	
	
	//Raw Min value for analog input
	{attribute 'OPC.UA.DA' :='1'}
	popa_0082_tt_3240_b_raw_min : REAL :=0;
	//Raw max value for analog input
	{attribute 'OPC.UA.DA' :='1'}
	popa_0082_tt_3240_b_raw_max : REAL :=32767;
	//EU Min value for analog input
	{attribute 'OPC.UA.DA' :='1'}
	popa_0082_tt_3240_b_eu_min : REAL;
	//EU Max value for analog input
	{attribute 'OPC.UA.DA' :='1'}
	popa_0082_tt_3240_b_eu_max : REAL;
	//Filter factor value for analog input
	{attribute 'OPC.UA.DA' :='1'}
	popa_0082_tt_3240_b_filter_factor : REAL;
	//Scaled value for analog input
	{attribute 'OPC.UA.DA' :='1'}
	popa_0082_tt_3240_b_scaled_value : REAL;
	
	//---tt_3340-----------------------------------------------------------------------------------------------------------------------
	//Alarm Priority setpoint
	{attribute 'OPC.UA.DA' :='1'}
	popa_0082_tt_3340_b_low_low_priority : INT;
	//Alarm delay setpoint(seconds)
	{attribute 'OPC.UA.DA' :='1'}
	popa_0082_tt_3340_b_low_low_delay_setpoint : INT;
	//Alarm active for HMI
	{attribute 'OPC.UA.DA' :='1'}
	popa_0082_tt_3340_b_low_low_active : BOOL;
	//Analog Alarm Setpoint
	{attribute 'OPC.UA.DA' :='1'}
	popa_0082_tt_3340_b_low_low_setpoint : REAL;
	//Alarm enable
	{attribute 'OPC.UA.DA' :='1'}
	popa_0082_tt_3340_b_low_low_enable: BOOL;
	
	//Alarm Priority setpoint
	{attribute 'OPC.UA.DA' :='1'}
	popa_0082_tt_3340_b_low_priority : INT;
	//Alarm delay setpoint(seconds)
	{attribute 'OPC.UA.DA' :='1'}
	popa_0082_tt_3340_b_low_delay_setpoint : INT;
	//Alarm active for HMI
	{attribute 'OPC.UA.DA' :='1'}
	popa_0082_tt_3340_b_low_active : BOOL;
	//Analog Alarm Setpoint
	{attribute 'OPC.UA.DA' :='1'}
	popa_0082_tt_3340_b_low_setpoint : REAL;
	//Alarm enable
	{attribute 'OPC.UA.DA' :='1'}
	popa_0082_tt_3340_b_low_enable: BOOL;
	
	//Alarm Priority setpoint
	{attribute 'OPC.UA.DA' :='1'}
	popa_0082_tt_3340_b_high_priority : INT;
	//Alarm delay setpoint(seconds)
	{attribute 'OPC.UA.DA' :='1'}
	popa_0082_tt_3340_b_high_delay_setpoint : INT;
	//Alarm active for HMI
	{attribute 'OPC.UA.DA' :='1'}
	popa_0082_tt_3340_b_high_active : BOOL;
	//Analog Alarm Setpoint
	{attribute 'OPC.UA.DA' :='1'}
	popa_0082_tt_3340_b_high_setpoint : REAL;
	//Alarm enable
	{attribute 'OPC.UA.DA' :='1'}
	popa_0082_tt_3340_b_high_enable: BOOL;
	
	//Alarm Priority setpoint
	{attribute 'OPC.UA.DA' :='1'}
	popa_0082_tt_3340_b_high_high_priority : INT;
	//Alarm delay setpoint(seconds)
	{attribute 'OPC.UA.DA' :='1'}
	popa_0082_tt_3340_b_high_high_delay_setpoint : INT;
	//Alarm active for HMI
	{attribute 'OPC.UA.DA' :='1'}
	popa_0082_tt_3340_b_high_high_active : BOOL;
	//Analog Alarm Setpoint
	{attribute 'OPC.UA.DA' :='1'}
	popa_0082_tt_3340_b_high_high_setpoint : REAL;
	//Alarm enable
	{attribute 'OPC.UA.DA' :='1'}
	popa_0082_tt_3340_b_high_high_enable: BOOL;
	
	
	//Raw Min value for analog input
	{attribute 'OPC.UA.DA' :='1'}
	popa_0082_tt_3340_b_raw_min : REAL :=0;
	//Raw max value for analog input
	{attribute 'OPC.UA.DA' :='1'}
	popa_0082_tt_3340_b_raw_max : REAL :=32767;
	//EU Min value for analog input
	{attribute 'OPC.UA.DA' :='1'}
	popa_0082_tt_3340_b_eu_min : REAL;
	//EU Max value for analog input
	{attribute 'OPC.UA.DA' :='1'}
	popa_0082_tt_3340_b_eu_max : REAL;
	//Filter factor value for analog input
	{attribute 'OPC.UA.DA' :='1'}
	popa_0082_tt_3340_b_filter_factor : REAL;
	//Scaled value for analog input
	{attribute 'OPC.UA.DA' :='1'}
	popa_0082_tt_3340_b_scaled_value : REAL;
	
	//---tt_3432-----------------------------------------------------------------------------------------------------------------------
	//Alarm Priority setpoint
	{attribute 'OPC.UA.DA' :='1'}
	popa_0092_tt_3432_b_low_low_priority : INT;
	//Alarm delay setpoint(seconds)
	{attribute 'OPC.UA.DA' :='1'}
	popa_0092_tt_3432_b_low_low_delay_setpoint : INT;
	//Alarm active for HMI
	{attribute 'OPC.UA.DA' :='1'}
	popa_0092_tt_3432_b_low_low_active : BOOL;
	//Analog Alarm Setpoint
	{attribute 'OPC.UA.DA' :='1'}
	popa_0092_tt_3432_b_low_low_setpoint : REAL;
	//Alarm enable
	{attribute 'OPC.UA.DA' :='1'}
	popa_0092_tt_3432_b_low_low_enable: BOOL;
	
	//Alarm Priority setpoint
	{attribute 'OPC.UA.DA' :='1'}
	popa_0092_tt_3432_b_low_priority : INT;
	//Alarm delay setpoint(seconds)
	{attribute 'OPC.UA.DA' :='1'}
	popa_0092_tt_3432_b_low_delay_setpoint : INT;
	//Alarm active for HMI
	{attribute 'OPC.UA.DA' :='1'}
	popa_0092_tt_3432_b_low_active : BOOL;
	//Analog Alarm Setpoint
	{attribute 'OPC.UA.DA' :='1'}
	popa_0092_tt_3432_b_low_setpoint : REAL;
	//Alarm enable
	{attribute 'OPC.UA.DA' :='1'}
	popa_0092_tt_3432_b_low_enable: BOOL;
	
	//Alarm Priority setpoint
	{attribute 'OPC.UA.DA' :='1'}
	popa_0092_tt_3432_b_high_priority : INT;
	//Alarm delay setpoint(seconds)
	{attribute 'OPC.UA.DA' :='1'}
	popa_0092_tt_3432_b_high_delay_setpoint : INT;
	//Alarm active for HMI
	{attribute 'OPC.UA.DA' :='1'}
	popa_0092_tt_3432_b_high_active : BOOL;
	//Analog Alarm Setpoint
	{attribute 'OPC.UA.DA' :='1'}
	popa_0092_tt_3432_b_high_setpoint : REAL;
	//Alarm enable
	{attribute 'OPC.UA.DA' :='1'}
	popa_0092_tt_3432_b_high_enable: BOOL;
	
	//Alarm Priority setpoint
	{attribute 'OPC.UA.DA' :='1'}
	popa_0092_tt_3432_b_high_high_priority : INT;
	//Alarm delay setpoint(seconds)
	{attribute 'OPC.UA.DA' :='1'}
	popa_0092_tt_3432_b_high_high_delay_setpoint : INT;
	//Alarm active for HMI
	{attribute 'OPC.UA.DA' :='1'}
	popa_0092_tt_3432_b_high_high_active : BOOL;
	//Analog Alarm Setpoint
	{attribute 'OPC.UA.DA' :='1'}
	popa_0092_tt_3432_b_high_high_setpoint : REAL;
	//Alarm enable
	{attribute 'OPC.UA.DA' :='1'}
	popa_0092_tt_3432_b_high_high_enable: BOOL;
	
	
	//Raw Min value for analog input
	{attribute 'OPC.UA.DA' :='1'}
	popa_0092_tt_3432_b_raw_min : REAL :=0;
	//Raw max value for analog input
	{attribute 'OPC.UA.DA' :='1'}
	popa_0092_tt_3432_b_raw_max : REAL :=32767;
	//EU Min value for analog input
	{attribute 'OPC.UA.DA' :='1'}
	popa_0092_tt_3432_b_eu_min : REAL;
	//EU Max value for analog input
	{attribute 'OPC.UA.DA' :='1'}
	popa_0092_tt_3432_b_eu_max : REAL;
	//Filter factor value for analog input
	{attribute 'OPC.UA.DA' :='1'}
	popa_0092_tt_3432_b_filter_factor : REAL;
	//Scaled value for analog input
	{attribute 'OPC.UA.DA' :='1'}
	popa_0092_tt_3432_b_scaled_value : REAL;
	
END_VAR

(* stored: Version 1.1.0.1, ProductVersion 3.1.4024.15
   GVL opc: Id {674fd3be-a48d-4a85-a2e2-bd0824412020} *)
